FUNCTION_BLOCK Pass50
  (* Standard: 61499-2 *)
  (* Version 0.1, 2017-00-01, hpea485, UOA *)
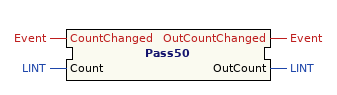
  EVENT_INPUT
    CountChanged;
  END_EVENT
  EVENT_OUTPUT
    OutCountChanged;
  END_EVENT
  VAR_INPUT
    Count : LINT;
  END_VAR
  VAR_OUTPUT
    OutCount : LINT;
  END_VAR
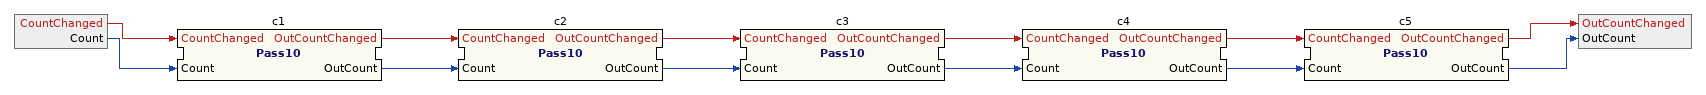
  FBS
    c1 : Pass10;
    c2 : Pass10;
    c3 : Pass10;
    c4 : Pass10;
    c5 : Pass10;
  END_FBS
  EVENT_CONNECTIONS
    CountChanged TO c1.CountChanged;
    c5.OutCountChanged TO OutCountChanged;
    c1.OutCountChanged TO c2.CountChanged;
    c2.OutCountChanged TO c3.CountChanged;
    c3.OutCountChanged TO c4.CountChanged;
    c4.OutCountChanged TO c5.CountChanged;
  END_CONNECTIONS
  DATA_CONNECTIONS
    Count TO c1.Count;
    c5.OutCount TO OutCount;
    c1.OutCount TO c2.Count;
    c2.OutCount TO c3.Count;
    c3.OutCount TO c4.Count;
    c4.OutCount TO c5.Count;
  END_CONNECTIONS
END_FUNCTION_BLOCK
